% RSLogix 500 project PLC Level 2 Project 7b.RSS, saved by version 8.30.00.16 %
PROJECT "UNTITLED"    % processor: Bul.1763 MicroLogix 1100 Series B %

PROGRAM FILES
  LAD 2 "MAIN"  4 rungs
  LAD 3 "IO CONFIG"  5 rungs
  LAD 4 "CTRL LOGIC"  7 rungs
  LAD 5 "CALI"  4 rungs

DATA FILES
  O0 OUTPUT  4 elements
  I1 INPUT  6 elements
  S2 STATUS  66 elements
  B3 BINARY  1 elements
  T4 TIMER  3 elements
  C5 COUNTER  2 elements
  R6 CONTROL  1 elements
  N7 INTEGER  6 elements
  F8 FLOAT  11 elements

LADDER 2 "MAIN"
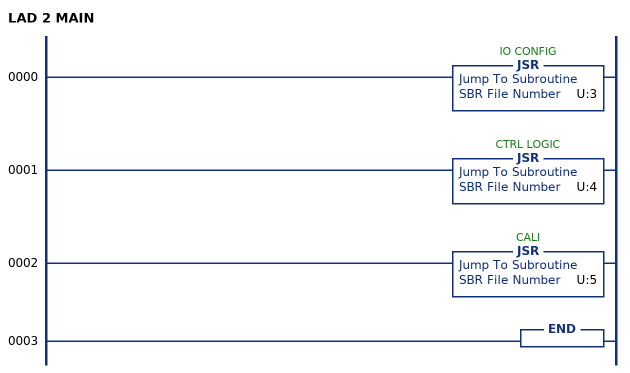
% Rung: 0 %
SOR JSR U:3 EOR
%   U:3  "IO CONFIG" %
% Rung: 1 %
SOR JSR U:4 EOR
%   U:4  "CTRL LOGIC" %
% Rung: 2 %
SOR JSR U:5 EOR
%   U:5  "CALI" %
% Rung: 3 %
SOR END EOR

LADDER 3 "IO CONFIG"
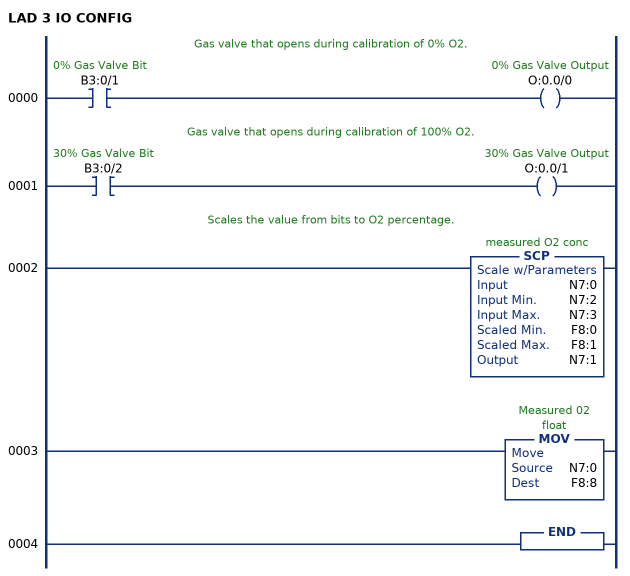
% Rung: 0 %
% Gas valve that opens during calibration of 0% O2. %
SOR XIC B3:0/1 OTE O:0.0/0 EOR
%   B3:0/1  "0% Gas Valve Bit" %
%   O:0.0/0  "0% Gas Valve Output" %
% Rung: 1 %
% Gas valve that opens during calibration of 100% O2. %
SOR XIC B3:0/2 OTE O:0.0/1 EOR
%   B3:0/2  "30% Gas Valve Bit" %
%   O:0.0/1  "30% Gas Valve Output" %
% Rung: 2 %
% Scales the value from bits to O2 percentage. %
SOR SCP N7:0 N7:2 N7:3 F8:0 F8:1 N7:1 EOR
%   N7:0  "02 sensor input signal" %
%   N7:2  "O2 input min" %
%   N7:3  "O2 input max" %
%   N7:1  "measured O2 conc" %
% Rung: 3 %
SOR MOV N7:0 F8:8 EOR
%   N7:0  "02 sensor input signal" %
%   F8:8  "Measured 02 float" %
% Rung: 4 %
SOR END EOR

LADDER 4 "CTRL LOGIC"
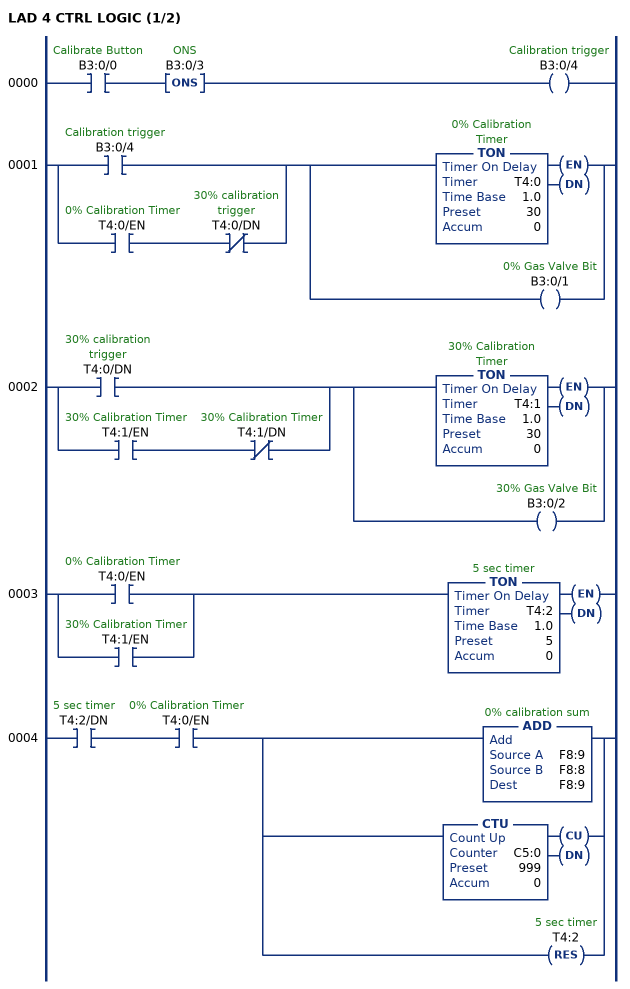
% Rung: 0 %
SOR XIC B3:0/0 ONS B3:0/3 OTE B3:0/4 EOR
%   B3:0/0  "Calibrate Button" %
%   B3:0/3  "ONS" %
%   B3:0/4  "Calibration trigger" %
% Rung: 1 %
SOR BST XIC B3:0/4 NXB XIC T4:0/EN XIO T4:0/DN BND BST TON T4:0 1.0 30 0 NXB OTE B3:0/1 BND EOR
%   B3:0/4  "Calibration trigger" %
%   T4:0  "0% Calibration Timer" %
%   T4:0/DN  "30% calibration trigger" %
%   B3:0/1  "0% Gas Valve Bit" %
% Rung: 2 %
SOR BST XIC T4:0/DN NXB XIC T4:1/EN XIO T4:1/DN BND BST TON T4:1 1.0 30 0 NXB OTE B3:0/2 BND EOR
%   T4:0/DN  "30% calibration trigger" %
%   T4:1  "30% Calibration Timer" %
%   B3:0/2  "30% Gas Valve Bit" %
% Rung: 3 %
SOR BST XIC T4:0/EN NXB XIC T4:1/EN BND TON T4:2 1.0 5 0 EOR
%   T4:0  "0% Calibration Timer" %
%   T4:1  "30% Calibration Timer" %
%   T4:2  "5 sec timer" %
% Rung: 4 %
SOR XIC T4:2/DN XIC T4:0/EN BST ADD F8:9 F8:8 F8:9 NXB CTU C5:0 999 0 NXB RES T4:2 BND EOR
%   T4:2  "5 sec timer" %
%   T4:0  "0% Calibration Timer" %
%   F8:9  "0% calibration sum" %
%   F8:8  "Measured 02 float" %

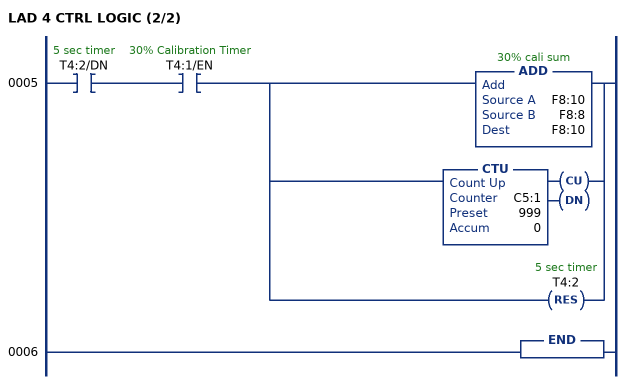
% Rung: 5 %
SOR XIC T4:2/DN XIC T4:1/EN BST ADD F8:10 F8:8 F8:10 NXB CTU C5:1 999 0 NXB RES T4:2 BND EOR
%   T4:2  "5 sec timer" %
%   T4:1  "30% Calibration Timer" %
%   F8:10  "30% cali sum" %
%   F8:8  "Measured 02 float" %
% Rung: 6 %
SOR END EOR

LADDER 5 "CALI"
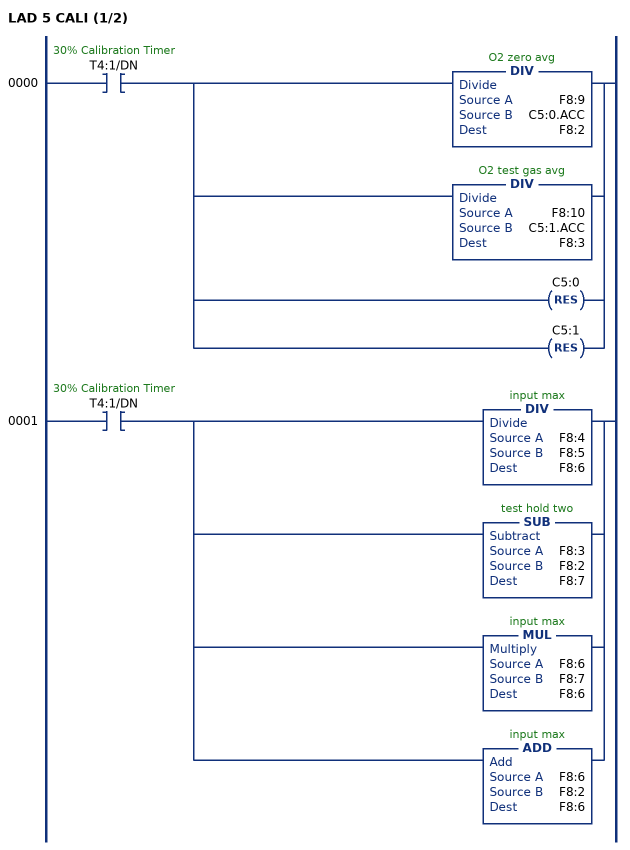
% Rung: 0 %
SOR XIC T4:1/DN BST DIV F8:9 C5:0.ACC F8:2 NXB DIV F8:10 C5:1.ACC F8:3 NXB RES C5:0 NXB RES C5:1 BND EOR
%   T4:1  "30% Calibration Timer" %
%   F8:9  "0% calibration sum" %
%   F8:2  "O2 zero avg" %
%   F8:10  "30% cali sum" %
%   F8:3  "O2 test gas avg" %
% Rung: 1 %
SOR XIC T4:1/DN BST DIV F8:4 F8:5 F8:6 NXB SUB F8:3 F8:2 F8:7 NXB MUL F8:6 F8:7 F8:6 NXB ADD F8:6 F8:2 F8:6 BND EOR
%   T4:1  "30% Calibration Timer" %
%   F8:4  "O2 max conc" %
%   F8:5  "O2 cali gas conc" %
%   F8:6  "input max" %
%   F8:3  "O2 test gas avg" %
%   F8:2  "O2 zero avg" %
%   F8:7  "test hold two" %

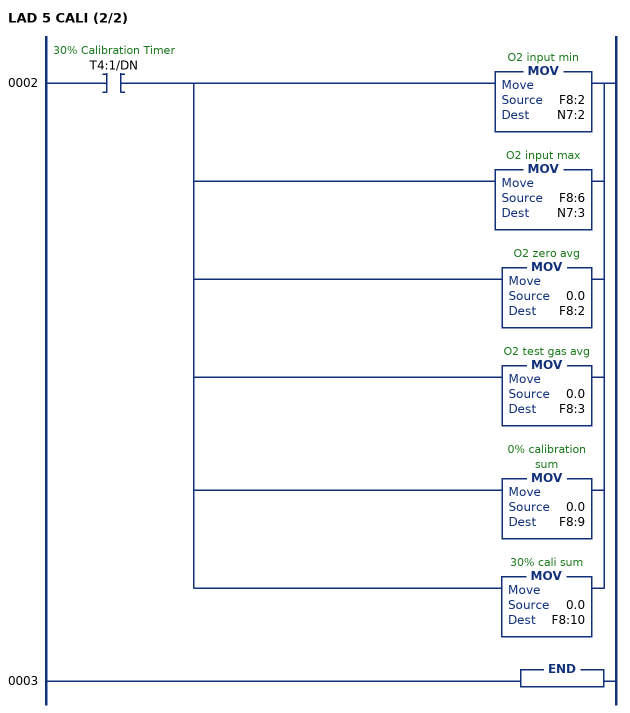
% Rung: 2 %
SOR XIC T4:1/DN BST MOV F8:2 N7:2 NXB MOV F8:6 N7:3 NXB MOV 0.0 F8:2 NXB MOV 0.0 F8:3 NXB MOV 0.0 F8:9 NXB MOV 0.0 F8:10 BND EOR
%   T4:1  "30% Calibration Timer" %
%   F8:2  "O2 zero avg" %
%   N7:2  "O2 input min" %
%   F8:6  "input max" %
%   N7:3  "O2 input max" %
%   F8:3  "O2 test gas avg" %
%   F8:9  "0% calibration sum" %
%   F8:10  "30% cali sum" %
% Rung: 3 %
SOR END EOR

OTHER DOCUMENTED ADDRESSES
  N7:4  "02 zero sum"
  N7:5  "O2 zero avg"

DATA TABLE (non-zero values as saved)
DATA T4
% .PRE .ACC %
% T4:0 % 30 0
% T4:1 % 30 0
% T4:2 % 5 0
DATA C5
% .PRE .ACC %
% C5:0 % 999 0
% C5:1 % 999 0
DATA N7
% N7:0 % 0 0 0 16383 0 0
DATA F8
% F8:0 % 0 40 0 0 40
% F8:5 % 30 0 0 0 0
